//Placeholder, WIP --> need to define what purpose this struct serves
TYPE ST_SafetyDiagnostics :
STRUCT
END_STRUCT
END_TYPE

(* stored: Version 1.1.0.1
   DUT ST_SafetyDiagnostics: Id {73cbece7-5a54-052a-2357-1389cfeaf33e} *)
